// TIA Portal V16 export
// export: Created 2026-03-31T12:43:18.3698547Z, ExportSetting WithDefaults, DisplayName Totally Integrated Automation Portal, DisplayVersion V16, DisplayName TIA Portal Version Control Interface, DisplayVersion V16, DisplayName TIA Portal Openness, DisplayVersion V16, DisplayName STEP 7 Professional, DisplayVersion V16, DisplayName STEP 7 Safety, DisplayVersion V16, DisplayName WinCC Advanced, DisplayVersion V16
VAR_GLOBAL   // PLC tag table "Default tag table"
   Mizga_ceh AT %I4.0 : Bool;
   Sok_flotweg AT %I4.1 : Bool;
   Voda_flotweg AT %I4.2 : Bool;
   Mizga_pr1 AT %I4.3 : Bool;
   Sok_pr1 AT %I4.4 : Bool;
   Voda_pr1 AT %I4.5 : Bool;
   Mizga_pr2 AT %I4.6 : Bool;
   Sok_pr2 AT %I4.7 : Bool;
   Voda_pr2 AT %I5.0 : Bool;
   Mizga_pr3 AT %I5.1 : Bool;
   Sok_pr3 AT %I5.2 : Bool;
   Voda_pr3 AT %I5.3 : Bool;
   Mizga_pr4 AT %I5.4 : Bool;
   Sok_pr4 AT %I5.5 : Bool;
   Voda_pr4 AT %I5.6 : Bool;
   "24_ok" AT %I5.7 : Bool;
   Blender AT %IW272 : Int;
   test_bool AT %I2.0 : Bool;
   T_Flotweg AT %IW274 : Int;
   Pastertizator_t AT %IW276 : Int;
   Blender_3 AT %IW278 : Int;
   fff AT %MW2 : Int;
   ffw AT %MW4 : Int;
   Reset_couter AT %M6.0 : Bool;
   Zero_blender AT %M6.1 : Bool;
   Valve_1 AT %Q11.0 : Bool;
   Valve_2 AT %Q11.1 : Bool;
   Valve_3 AT %Q11.2 : Bool;
   Valve_4 AT %Q11.3 : Bool;
   Valve_5 AT %Q11.4 : Bool;
   Valve_6 AT %Q11.5 : Bool;
   Valve_7 AT %Q11.6 : Bool;
   Valve_8 AT %Q11.7 : Bool;
   Speed_pump_prod AT %QW288 : Int;
   M1_product AT %Q12.0 : Bool;
   M3_Water AT %Q12.1 : Bool;
   Temp_paster AT %MW50 : Int;
   Test_HMI AT %M40.0 : Bool;
   Damp_valve_out_up AT %Q12.2 : Bool;
   Damp_valve_out_down AT %Q12.3 : Bool;
   IW_Tank3 AT %IW10 : Int;
   IW_Tank4 AT %IW12 : Int;
   IW_Tank5 AT %IW14 : Int;
   IW_Tank6 AT %IW16 : Int;
   IW_Tank7 AT %IW20 : Int;
   IW_Tank8 AT %IW22 : Int;
   IW_Tank9 AT %IW24 : Int;
   IW_Tank10 AT %IW26 : Int;
   IW_Tank11 AT %IW30 : Int;
   IW_Tank12 AT %IW32 : Int;
   IW_Tank13 AT %IW34 : Int;
   IW_Tank14 AT %IW36 : Int;
   tag_1 AT %M0.1 : Bool;
END_VAR
